FUNCTION_BLOCK SimpleNOT (* NOT for boolean *)
  (* Standard: 61499-1; Description: Copyright (c) 2023 Johannes Kepler University Linz This program and the accompanying materials are made available under the terms of the Eclipse Public License 2.0 which is available at https://www.eclipse.org/legal/epl-2.0/ SPDX-License-Identifier: EPL-2.0 *)
  (* Version 1.0, 2022-08-30, Bianca Wiesmayr, Johannes Kepler University Linz, initial API and implementation and/or initial documentation *)
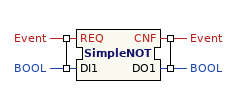
  EVENT_INPUT
    REQ WITH DI1; (* Normal Execution Request *)
  END_EVENT
  EVENT_OUTPUT
    CNF WITH DO1; (* Execution Confirmation *)
  END_EVENT
  VAR_INPUT
    DI1 : BOOL;
  END_VAR
  VAR_OUTPUT
    DO1 : BOOL;
  END_VAR
  ALGORITHM REQ IN ST:
	DO1 := NOT DI1;
  END_ALGORITHM
END_FUNCTION_BLOCK
